# EPICS autosave request: CARSApp/Db/sca_window.req
# FILE...
$(P)$(SCA):WIN.VAL
$(P)$(SCA):LLD.VAL
$(P)$(SCA):WIN_tweakVal.VAL
$(P)$(SCA):LLD_tweakVal.VAL
